{attribute 'qualified_only'}
{attribute 'strict'}
{attribute 'to_string'}
// Drive states based on the CiA402 state machine
TYPE E_L7NHA_DriveState :
(
	SWITCH_ON_DISABLED,
	READY_TO_SWITCH_ON,
	SWITCHED_ON,
	OPERATION_ENABLED,
	QUICK_STOP_ACTIVE,
	FAULT_REACTION_ACTIVE,
	FAULT
);
END_TYPE

(* stored: Version 1.1.0.1, ProductVersion 3.1.4024.15
   DUT E_L7NHA_DriveState: Id {abfcfe37-791d-41ec-b716-3c934062ed26} *)
